(* CoDeSys 2.3 project: skv_owen1.6.pro *)
(* Title: Контроль и управление скважинами. *)
(* Version: 1.6 *)
(* Author: Пичугин А.В. *)
(* Description: Автоматизированная система контроля и управления
водонасосной станции Печорского ЛПУ МГ *)
(* Libraries: STANDARD.LIB 4.10.05 11:14:46, IECSFC.LIB 13.4.06 15:51:28, SYSLIBTIME.LIB 20.2.06 13:31:16, SysLibMem.lib 20.2.06 13:31:12, SysLibCom.lib 20.2.06 13:31:08, SYSTASKINFO.LIB 20.2.06 13:31:38, ANALYZATION.LIB 5.10.99 09:05:06, SYSLIBCALLBACK.LIB 20.2.06 13:31:08, Util.lib 18.5.10 15:14:28 *)

(* PLC configuration (modules and I/O channels)
Discrete input 8 bit [ID100] node 0, in %IB0 out %QB0 {Filtrationtime = 10; Filtrationtime = 10; Filtrationtime = 10; Filtrationtime = 10; Filtrationtime = 10; Filtrationtime = 10; Filtrationtime = 10; Filtrationtime = 10; Visibility = Yes; PinCount = 8; WatchDogPeriod = 1000; PollPeriod = 1}
  AT %IB0.0 [ByteInput] 8 discrete inputs
Discrete output - relay [ID102] node 1, in %IB1 out %QB1 {PinCount = 1; SafeValueBool = FALSE; Visibility = Yes}
  Pump4_block AT %QX1.0 [BitOutput] Блокировка насоса 4 (relay)
Discrete output - relay [ID102] node 2, in %IB2 out %QB2 {PinCount = 1; SafeValueBool = FALSE; Visibility = Yes}
  Pump5_block AT %QX2.0 [BitOutput] Блокировка насоса 5 (relay)
Discrete output - relay [ID102] node 3, in %IB3 out %QB3 {PinCount = 1; SafeValueBool = FALSE; Visibility = No}
  AT %QX3.0 [BitOutput] relay
Discrete output - relay [ID102] node 4, in %IB4 out %QB4 {PinCount = 1; SafeValueBool = FALSE; Visibility = No}
  AT %QX4.0 [BitOutput] relay
Discrete output - relay [ID102] node 5, in %IB5 out %QB5 {PinCount = 1; SafeValueBool = FALSE; Visibility = No}
  AT %QX5.0 [BitOutput] relay
Discrete output - relay [ID102] node 6, in %IB6 out %QB6 {PinCount = 1; SafeValueBool = FALSE; Visibility = No}
  AT %QX6.0 [BitOutput] relay
Special output [ID104] node 7, in %IB7 out %QB7 {Visibility = No; PinCount = 1}
  AT %QX7.0 [BitOutput] Special output
Owen (Master) [OWEN_MASTER_ID451] node 8, in %IB8 out %QB8 {Timeout = 50; Visibility = Yes}
  LError AT %QW8.0 [WordOutput] Last error
  AT %QW8.1 [WordOutput] Last hash
  LAddress AT %QW8.2 [WordOutput] Last address
  AT %QB8.3 [ComChannel] Start/Stop)
  RS-485-1 [COM1_USART] node 0, in %IB8.0 out %QB8.0 {CommunicationSpeed = 11520; Parity = NO PARITY CHECK; BitLength = 8 bits; StopLength = One stop bit; InterfaceType = RS485; FrameOriented = ASCII; Timeout = 0; Visibility = Yes}
Box_Temp AT %QD8.1.0 [FloatOutput] Температура внутренняя
Outbox_Temp AT %QD8.2.0 [FloatOutput] Температура наружная
Skv4_Temp AT %QD8.3.0 [FloatOutput] Температура внутренняя
Skv4_Level AT %QD8.4.0 [FloatOutput] Уровень воды
Skv5_Temp AT %QD8.5.0 [FloatOutput] Температура внутренняя
Skv5_Level AT %QD8.6.0 [FloatOutput] Уровень воды
Skv4_level_alarm AT %QD8.7.0 [FloatOutput] Блокировка насоса
Skv5_level_alarm AT %QD8.8.0 [FloatOutput] Блокировка насоса
Skv4_Counter AT %QD8.9.0.0 [DWordOutput] Текущее значение счетчика
Skv5_Counter AT %QD8.10.0.0 [DWordOutput] Текущее значение счетчика
Skv4_Rate AT %QD8.11.0.0 [DWordOutput] Текущее значение счетчика в физических величинах
Skv5_Rate AT %QD8.12.0.0 [DWordOutput] Текущее значение счетчика в физических величинах
Skv4_dec AT %QW8.13.0.0 [WordOutput] Положение десятичной точки умножителя
Skv5_dec AT %QW8.14.0.0 [WordOutput] Положение десятичной точки умножителя
Max_temp AT %ID9.0 [FloatInput] Максимальная температура
Min_temp AT %ID10.0 [FloatInput] Минимальная температура
Max_level AT %ID11.0 [FloatInput] Верхний аварийный уровень (ВАУ)
*)

(* Task configuration *)
TASK Alarm_control (PRIORITY := 1, INTERVAL := T#1000ms);
	Alarm_control();
END_TASK
TASK Alarm_rate_control (PRIORITY := 1, INTERVAL := T#20000ms);
	Alarm_rate_control();
END_TASK
TASK Main (PRIORITY := 1, INTERVAL := T#100ms);
	PLC_PRG();
END_TASK
TASK Terminal (PRIORITY := 1, INTERVAL := T#50ms);
	Terminal();
END_TASK

(* Global variable list: Global_Variables *)
VAR_GLOBAL RETAIN
	SMS_sPhone:ARRAY[0..4] OF STRING :='','','','','+79225830093';  				(*Номера телефонов*)
	SMS_bPhone_info:ARRAY[0..4] OF BOOL:=FALSE,FALSE,FALSE,FALSE,TRUE;		(*Отсылать ли на соотв. телефон информацию*)
	SMS_bPhone_alarm:ARRAY[0..4] OF BOOL:=FALSE,FALSE,FALSE,FALSE,TRUE;	(*Отсылать ли на соотв. телефон аварии*)
	bAlarm_old:ARRAY[0..15] OF BOOL;
	iTime_info:INT:=12; (*Время отправки информации*)
	sBalance:STRING(255);
	bRateControl:BOOL:=FALSE; (*будем считать расход?*)
END_VAR

(* Global variable list: Other *)
VAR_GLOBAL
	bAlarm:ARRAY[0..15] OF BOOL; (*Аварии текущие по 1 на каждую аварию.*)
	bAlarm_send:ARRAY[0..15] OF BOOL; (*Необходимость посылки сообщения об аварии по 1 на каждую аварию.*)
	Message:ARRAY[0..15] OF STRING; (*Сообщения о появлении или исчезновении аварий*)
	bRun:BOOL; (*Разрешение на запуск*)
	tRun:TON; (*таймер задержки начала работы*)
	(*Max_temp:REAL:=45; Максимальная температура в боксе*)
	(*Min_temp:REAL:=3; Минимальная температура в боксе*)
	rHist_temp:REAL:=1; (*Гистерезис температуры*)
	(*Max_level:REAL:=73; Верхний аварийный уровень (ВАУ)*)
	Min_level:REAL:=3; (*Нижний аварийный уровень (НАУ)*)
	rHist_level:REAL:=1; (*Гистерезис уровня*)

END_VAR

(* Global variable list: Text *)
VAR_GLOBAL
	a0:STRING:='ALARM!$0D$0A Skv4 Low Level$0D$0A Pump BLOCK $0D$0A';
	n0:STRING:='NORMA.$0D$0A Skv4 Normal Level$0D$0A Pump READY $0D$0A';
	a1:STRING:='ALARM!$0D$0A Skv5 Low Level$0D$0A Pump BLOCK $0D$0A';
	n1:STRING:='NORMA.$0D$0A Skv5 Normal Level$0D$0A Pump READY $0D$0A';
	a2:STRING:='ALARM!$0D$0A Skv4 High Level $0D$0A';
	n2:STRING:='NORMA.$0D$0A Skv4 Normal Level $0D$0A';
	a3:STRING:='ALARM!$0D$0A Skv5 High Level $0D$0A';
	n3:STRING:='NORMA.$0D$0A Skv5 Normal Level $0D$0A';
	a4:STRING:='ALARM!$0D$0A Skv4 No Flow $0D$0A';
	n4:STRING:='NORMA.$0D$0A Skv4 Flow On $0D$0A';
	n41:STRING:='NORMA.$0D$0A Skv4 Flow Off $0D$0A';
	a5:STRING:='ALARM!$0D$0A Skv5 No Flow $0D$0A';
	n5:STRING:='NORMA.$0D$0A Skv5 Flow On $0D$0A';
	n51:STRING:='NORMA.$0D$0A Skv5 Flow Off $0D$0A';
	a6:STRING:='ALARM!$0D$0A Skv4 Low Temperature $0D$0A';
	n6:STRING:='NORMA.$0D$0A Skv4 Normal Temperature $0D$0A';
	a7:STRING:='ALARM!$0D$0A Skv5 Low Temperature $0D$0A';
	n7:STRING:='NORMA.$0D$0A Skv5 Normal Temperature $0D$0A';
	a8:STRING:='ALARM!$0D$0A Box Low Temperature $0D$0A';
	n8:STRING:='NORMA.$0D$0A Box Normal Temperature $0D$0A';
	a9:STRING:='ALARM!$0D$0A Skv4 High Temperature $0D$0A';
	n9:STRING:='NORMA.$0D$0A Skv4 Normal Temperature $0D$0A';
	a10:STRING:='ALARM!$0D$0A Skv5 High Temperature $0D$0A';
	n10:STRING:='NORMA.$0D$0A Skv5 Normal Temperature $0D$0A';
	a11:STRING:='ALARM!$0D$0A Box High Temperature $0D$0A';
	n11:STRING:='NORMA.$0D$0A Box Normal Temperature $0D$0A';
	a12:STRING:='ALARM!$0D$0A Skv4 No Link $0D$0A';
	n12:STRING:='NORMA.$0D$0A Skv4 Link on $0D$0A';
	a13:STRING:='ALARM!$0D$0A Skv5 No Link $0D$0A';
	n13:STRING:='NORMA.$0D$0A Skv5 Link on $0D$0A';
	a14:STRING:='ALARM!$0D$0A Box No Link $0D$0A';
	n14:STRING:='NORMA.$0D$0A Box Link on $0D$0A';
	a15:STRING:='ALARM!$0D$0A Box No Power $0D$0A';
	n15:STRING:='NORMA.$0D$0A Box Power on $0D$0A';
END_VAR

(* POU Alarm_control, ST *)
PROGRAM Alarm_control
VAR
(*Обработка гвоздей, грызунов, монтажников, и солнечного затмения*)
	er_72: Get_Modules_Errors; (*адрес 9, ТРМ202 в боксе*)
	er_88: Get_Modules_Errors; (*адрес 11, ТРМ202 скважина 4*)
	er_104: Get_Modules_Errors; (*адрес 13, СИ30 скважина 4*)
	er_112: Get_Modules_Errors; (*адрес 14, ТРМ202 скважина 5*)
	er_128: Get_Modules_Errors; (*адрес 16, СИ30 скважина 5*)
(*Каждому модулю даем свою ошибку*)
	mod_72:BOOL:=0; (* 1 - если ошибка связи, 0 - нет *)
	mod_88:BOOL:=0;  (* 1 - если ошибка связи, 0 - нет *)
	mod_104:BOOL:=0;  (* 1 - если ошибка связи, 0 - нет *)
	mod_112:BOOL:=0;  (* 1 - если ошибка связи, 0 - нет *)
	mod_128:BOOL:=0;  (* 1 - если ошибка связи, 0 - нет *)
	hist_tempb_min:HIST;
	hist_tempb_max:HIST;
	hist_temp4_min:HIST;
	hist_temp4_max:HIST;
	hist_temp5_min:HIST;
	hist_temp5_max:HIST;
	hist_level4:HIST;
	hist_level5:HIST;
	tempb_max: BOOL;
	tempb_min: BOOL;
	temp4_max: BOOL;
	temp5_max: BOOL;
	temp5_min: BOOL;
	temp4_min: BOOL;
	level5: BOOL;
	level4: BOOL;
END_VAR
IF NOT bRun THEN
	RETURN;
END_IF

IF NOT mod_88 THEN (*если нет ошибки связи  с ТРМ202 скважина 4*)
	IF Skv4_level_alarm>0 THEN (*Проверка аварии Скв4 НАУ *)
		bAlarm[0] := TRUE;
		Message[0]:=a0;
	ELSE
		bAlarm[0] := FALSE;
		Message[0]:=n0;
	END_IF
(*-----------------------------------------------------------------------------------------------------------*)
	hist_level4(LOW:=REAL_TO_INT(Max_level-rHist_level), HIGH:=REAL_TO_INT(Max_level+rHist_level), IN:=REAL_TO_INT(Skv4_Level), OUT=>level4);
	IF  level4 THEN (*Проверка аварии Скв4 ВАУ *)
		bAlarm[2] := TRUE;
		Message[2]:=a2;
	ELSE
		bAlarm[2] := FALSE;
		Message[2]:=n2;
	END_IF
(*-----------------------------------------------------------------------------------------------------------*)
	hist_temp4_min(LOW:=REAL_TO_INT(Min_temp-rHist_temp), HIGH:=REAL_TO_INT(Min_temp+rHist_temp), IN:=REAL_TO_INT(Skv4_Temp), OUT=>temp4_min);
	IF  NOT temp4_min THEN (*Проверка аварии Скв4 темп. ниже нормы *)
		bAlarm[6] := TRUE;
		Message[6]:=a6;
	ELSE
		bAlarm[6] := FALSE;
		Message[6]:=n6;
	END_IF
(*-----------------------------------------------------------------------------------------------------------*)
	hist_temp4_max(LOW:=REAL_TO_INT(Max_temp-rHist_temp), HIGH:=REAL_TO_INT(Max_temp+rHist_temp), IN:=REAL_TO_INT(Skv4_Temp), OUT=>temp4_max);
	IF  temp4_max THEN (*Проверка аварии Скв4 темп. выше нормы *)
		bAlarm[9] := TRUE;
		Message[9]:=a9;
	ELSE
		bAlarm[9] := FALSE;
		Message[9]:=n9;
	END_IF
END_IF
(*-----------------------------------------------------------------------------------------------------------*)
(*-----------------------------------------------------------------------------------------------------------*)
IF NOT mod_112 THEN (*если нет ошибки связи  с ТРМ202 скважина 5*)
	IF Skv5_level_alarm>0 THEN  (*Проверка аварии Скв5 НАУ*)
		bAlarm[1] := TRUE;
		Message[1]:=a1;
	ELSE
		bAlarm[1] := FALSE;
		Message[1]:=n1;
	END_IF
(*-----------------------------------------------------------------------------------------------------------*)
	hist_level5(LOW:=REAL_TO_INT(Max_level-rHist_level), HIGH:=REAL_TO_INT(Max_level+rHist_level), IN:=REAL_TO_INT(Skv5_Level), OUT=>level5);
	IF level5 THEN (*Проверка аварии Скв5 ВАУ *)
		bAlarm[3] := TRUE;
		Message[3]:=a3;
	ELSE
		bAlarm[3] := FALSE;
		Message[3]:=n3;
	END_IF
(*-----------------------------------------------------------------------------------------------------------*)
	hist_temp5_min(LOW:=REAL_TO_INT(Min_temp-rHist_temp), HIGH:=REAL_TO_INT(Min_temp+rHist_temp), IN:=REAL_TO_INT(Skv5_Temp), OUT=>temp5_min);
	IF  NOT temp5_min THEN (*Проверка аварии Скв5 темп. ниже нормы *)
		bAlarm[7] := TRUE;
		Message[7]:=a7;
	ELSE
		bAlarm[7] := FALSE;
		Message[7]:=n7;
	END_IF
(*-----------------------------------------------------------------------------------------------------------*)
	hist_temp5_max(LOW:=REAL_TO_INT(Max_temp-rHist_temp), HIGH:=REAL_TO_INT(Max_temp+rHist_temp), IN:=REAL_TO_INT(Skv5_Temp), OUT=>temp5_max);
	IF   temp5_max THEN (*Проверка аварии Скв5 темп. выше нормы *)
		Message[10]:=a10;
		bAlarm[10] := TRUE;
	ELSE
		bAlarm[10] := FALSE;
		Message[10]:=n10;
	END_IF
END_IF
(*-----------------------------------------------------------------------------------------------------------*)
(*Аварии Нет протока определяются отдельно в программе Alarm_rate_control *)
(*-----------------------------------------------------------------------------------------------------------*)

IF NOT mod_72 THEN (*если нет ошибки связи  с ТРМ202 щитовая*)
	hist_tempb_min(LOW:=REAL_TO_INT(Min_temp-rHist_temp), HIGH:=REAL_TO_INT(Min_temp+rHist_temp), IN:=REAL_TO_INT(Box_Temp), OUT=>tempb_min);
	IF  NOT tempb_min THEN (*Проверка аварии Щит.  темп. ниже нормы *)
		bAlarm[8] := TRUE;
		Message[8]:=a8;
	ELSE
		bAlarm[8] := FALSE;
		Message[8]:=n8;
	END_IF
(*-----------------------------------------------------------------------------------------------------------*)
	hist_tempb_max(LOW:=REAL_TO_INT(Max_temp-rHist_temp), HIGH:=REAL_TO_INT(Max_temp+rHist_temp), IN:=REAL_TO_INT(Box_Temp), OUT=>tempb_max);
	IF  tempb_max THEN (*Проверка аварии Щит. темп. выше нормы *)
		bAlarm[11] := TRUE;
		Message[11]:=a11;
	ELSE
		bAlarm[11] := FALSE;
		Message[11]:=n11;
	END_IF
END_IF
(*-----------------------------------------------------------------------------------------------------------*)
(*-----------------------------------------------------------------------------------------------------------*)
(*Аварии Нет связи определяются  в программе Get_Modules_Errors *)
CASE LAddress OF
	72:
		er_72(err:=LError , stat=> mod_72);
	88:
		er_88(err:=LError , stat=> mod_88);
	104:
		er_104(err:=LError , stat=> mod_104);
	112:
		er_112(err:=LError , stat=> mod_112);
	128:
		er_128(err:=LError , stat=> mod_128);
END_CASE;

IF  mod_88 OR mod_104 THEN (*Проверка аварии Нет связи с скв. 4 *)
	bAlarm[12] := TRUE;
	Message[12]:=a12;
ELSE
	bAlarm[12] := FALSE;
	Message[12]:=n12;
END_IF

IF  mod_112 OR mod_128 THEN (*Проверка аварии Нет связи с скв. 5 *)
	bAlarm[13] := TRUE;
	Message[13]:=a13;
ELSE
	bAlarm[13] := FALSE;
	Message[13]:=n13;
END_IF

IF  mod_72 THEN (*Проверка аварии Нет связи с щит. *)
	bAlarm[14] := TRUE;
	Message[14]:=a14;
ELSE
	bAlarm[14] := FALSE;
	Message[14]:=n14;
END_IF

(*-----------------------------------------------------------------------------------------------------------*)
IF V220_enable=FALSE THEN  (*Проверка аварии нет питания *)
	bAlarm[15] := TRUE;
	Message[15]:=a15;
ELSE
	bAlarm[15] := FALSE;
	Message[15]:=n15;
END_IF;

(*-------------------------А теперь управляем!-------------------------------------------------*)
IF bAlarm[0] OR bAlarm[4] THEN
	Pump4_block := TRUE;
ELSE
	Pump4_block := FALSE;
END_IF
IF bAlarm[1] OR bAlarm[5] THEN
	Pump5_block := TRUE;
ELSE
	Pump5_block := FALSE;
END_IF
END_PROGRAM

(* POU Get_Modules_Errors, ST *)
FUNCTION_BLOCK Get_Modules_Errors
VAR_INPUT
	err:WORD;
END_VAR
VAR_OUTPUT
	stat:BOOL:=0;
END_VAR
VAR
	bErr:BOOL;
	rt: R_TRIG;
	tim_err: TIME := T#5s;
	t: TON;
END_VAR
IF err=81 THEN
	bErr:=TRUE;
ELSE
	bErr:=FALSE;
END_IF
(*Тригер прихода ошибки*)
rt(CLK:=bErr);
(*Если пришла ошибка, запускаем таймер*)
IF rt.Q THEN
	t(IN:=TRUE , PT:=tim_err);
END_IF
(*Вызываем таймер*)
t;
(*Если таймер не запущен и ошибки нет, то аварии нет*)
IF t.IN=FALSE AND NOT bErr THEN
	stat:=FALSE;
END_IF
(*Если таймер запущен, а ошибка ушла, то была помеха, отключаем аварию и таймер*)
IF t.IN AND err=0 THEN
	t(IN:=FALSE , PT:=tim_err);
	stat:=FALSE;
END_IF
(*Если таймер отработал, а ошибка не ушла - беда, ищем ваши гвозди ))) *)
IF t.Q THEN
	stat:=TRUE;
	t(IN:=FALSE , PT:=tim_err);
END_IF

RETURN;
END_FUNCTION_BLOCK

(* POU HIST, ST *)
FUNCTION_BLOCK HIST
VAR_INPUT
	IN:REAL;
	HIGH:REAL;
	LOW:REAL;
END_VAR
VAR_OUTPUT
	OUT:BOOL;
END_VAR
VAR
END_VAR
IF IN>HIGH THEN
	OUT:=TRUE;
END_IF
IF IN<LOW THEN
	OUT:=FALSE;
END_IF
END_FUNCTION_BLOCK

(* POU Alarm_rate_control, ST *)
PROGRAM Alarm_rate_control
VAR
	Skv4_tmp:DWORD;
	Skv5_tmp:DWORD;
END_VAR
IF NOT bRun THEN
	RETURN;
END_IF

IF bRateControl THEN
	IF Pump4_on THEN
		IF Skv4_Counter <> Skv4_tmp THEN
			bAlarm[4]:=FALSE;
			Message[4]:=n4;
			Skv4_tmp :=Skv4_Counter;
		ELSE
			bAlarm[4] := TRUE;
			Message[4]:=a4;
		END_IF;
	ELSE
		bAlarm[4] := FALSE;
		Message[4]:=n41;
		Skv4_tmp:=0;
	END_IF


	IF Pump5_on THEN
		IF Skv5_Counter <> Skv5_tmp THEN
			bAlarm[5] := FALSE;
			Message[5]:=a5;
			Skv5_tmp :=Skv5_Counter;
		ELSE
			bAlarm[5] := TRUE;
			Message[4]:=n5;
		END_IF
	ELSE
		bAlarm[5] := FALSE;
		Message[5]:=n51;
		Skv5_tmp:=0;
	END_IF
ELSE
	bAlarm[4]:= FALSE;
	bAlarm[5]:= FALSE;
END_IF
END_PROGRAM

(* POU PLC_PRG, ST *)
PROGRAM PLC_PRG
VAR
	SMS_txt: STRING(255) := '';					(*Сформированый текст СМС*)
	SMS_txt_tip:INT:=1;						(*Тип СМС. 1-аварии, 2-информация, 3-разное*)
	must_send_sms:BOOL:=FALSE;		(*Признак необходимости отправить СМС*)
	bPhone_send:ARRAY[0..4] OF BOOL:=FALSE,FALSE,FALSE,FALSE,FALSE;
	FB_SMS:GSM_Modem_SMS;
	i:INT:=0;										(*для счетчиков*)
	j:INT:=0;										(*для счетчиков*)
	jj:INT:=0;										(*для счетчиков*)
	tmp_num:STRING;
	tmp_ind:INT;
	sBalanceNum:STRING:='111';
	sBalanceText:STRING:='11';
	sBalanceCom:STRING:='AT+CUSD=1,"#100#"$0D$0A';
	com_num:PORTS:=COM1;
	sInput_command1:STRING:='Replace phone'; (*Команда смены номера телефона*)
	sInput_command2:STRING:='Alarm on'; (*Команда включения посылки аварий на телефон*)
	sInput_command3:STRING:='Alarm off'; (*Команда отключения посылки аварий на телефон*)
	sInput_command4:STRING:='Info on'; (*Команда включения посылки информации на телефон*)
	sInput_command5:STRING:='Info off'; (*Команда отключения посылки информации на телефон*)
	sInput_command6:STRING:='Get info'; (*Команда получения информации на телефон*)
	sInput_command7:STRING:='Get alarm'; (*Команда получения аварий на телефон*)
	sInput_command8:STRING:='Set time'; (*Команда установки времени отправки информации на телефоны*)
	sInput_command9:STRING:='Rate on'; (*Команда включения проверки аварии нет протока*)
	sInput_command10:STRING:='Rate off'; (*Команда выключения проверки аварии нет протока*)
	rSkv4_Rate_dec: REAL;
	rSkv5_Rate_dec: REAL;
	bInfoSended: BOOL:=FALSE; (*признак того, что информация уже отослана*)
	bBalanseQ: BOOL; (*признак запроса баланса*)
END_VAR
IF NOT bRun THEN
tRun(IN := TRUE , PT:= T#3s);
END_IF
tRun;
IF  tRun.Q THEN
	tRun(IN := FALSE, PT:= T#3s);
	SysMemSet (ADR(bAlarm_old),16#00,SIZEOF(bAlarm_old)); (*Заполняем массив отправленых аварий 0-ми, теперь все аварии станут новыми*)
	bRun:=TRUE;
END_IF
IF NOT bRun THEN
	RETURN;
END_IF


 IF must_send_sms THEN (*Если необходимо послать СМС вызываем ФБ в цикле непрерывно пока не будет выставлен выход ФБ GSM_Modem_SMS sended_OK*)
 (*********************отправляем СМС всем из списка, с учетом фильтра bPhone_send*****************************)

	CASE i OF (*перебираем телефоны*)
	0..4:	IF bPhone_send[i] AND LEN(SMS_sPhone[i])>0 THEN (*если телефону разрешено получать  и он не пустой*)
				fb_sms(com_num:=COM1,phone_num:=SMS_sPhone[i],send_SMS_text:=SMS_txt ,rcvSMS:=FALSE ); (*отправляем*)
					IF fb_sms.sended_OK THEN (*когда отправлено, переключаемся на следующий телефон*)
						IF bPhone_send[0]=TRUE THEN (*если была разрешена отправка на 0 телефон, то дальше перебирать не надо*)
							i:=255;
						ELSE
							i:=i+1;
						END_IF
					ELSE
						i:=i;
					END_IF
			ELSE (* если не разрешено, просто переключаемся на следующий телефон*)
				i:=i+1;
			END_IF
	ELSE   (* телефоны кончились, всё на родину*)
		i:=0;
		SMS_sPhone[0]:='';
		bPhone_send[0]:=FALSE; (*запрещаем посылку*)
		bPhone_send[1]:=FALSE;
		bPhone_send[2]:=FALSE;
		bPhone_send[3]:=FALSE;
		bPhone_send[4]:=FALSE;
		must_send_sms:=FALSE;


		IF  SMS_txt_tip=1 THEN
			bAlarm_old[jj]:=bAlarm[jj]; (*и отмечаем, что на аварию отреагировали*)
		END_IF
	END_CASE


(******************************************************************************************************)
(******************************************************************************************************)
ELSE (*Иначе - просто проверяем полученные  смс и следим за авариями *)


	fb_sms(com_num:=COM1,phone_num:='',send_SMS_text:='' ,rcvSMS:=TRUE );

(******************Проверяем команду на замену номера телефона***********************)
	IF FIND(fb_sms.rcvedSMS,sInput_command1)>0 THEN
		tmp_ind:=STRING_TO_INT(MID(fb_sms.rcvedSMS,1,15));
		tmp_num:=MID(fb_sms.rcvedSMS,12,17);
		IF tmp_ind>=1 AND tmp_ind<=4 THEN (*если индекс от 1 до 4, то выполняем*)
			SMS_txt:=sGetTime(0);
			SMS_txt:=CONCAT('Replace ',SMS_sPhone[tmp_ind]); (*готовим подтверждающую СМС*)
			SMS_txt:=CONCAT(SMS_txt,' on '); (*готовим*)
			SMS_txt:=CONCAT(SMS_txt,tmp_num); (*готовим*)
			SMS_txt:=CONCAT(SMS_txt,' OK '); (*готово*)
			SMS_sPhone[tmp_ind]:=tmp_num; (*меняем номер*)
		ELSE
			SMS_txt:='Error! Index mast be from 1 to 4'; (*если индекс не верен, то СМС с ошибкой*)
		END_IF
		SMS_txt_tip:=3; (*тип СМС - разное*)
		SMS_sPhone[0]:=fb_sms.rcvedPhonNum; (*номер для ответа - тот с которого пришла команда*)
		bPhone_send[0]:=TRUE;
		must_send_sms:=TRUE; (*включаем отправку*)
		RETURN; (*уходим на отправку*)
	END_IF
(******************************************************************************************************)
(******************Проверяем команду на включение посылки аварий на телефон***********************)
	IF FIND(fb_sms.rcvedSMS,sInput_command2)>0 AND iIsPhone(fb_sms.rcvedPhonNum)>0THEN
		SMS_bPhone_alarm[iIsPhone(fb_sms.rcvedPhonNum)]:=TRUE;
		SMS_txt:=CONCAT(sGetTime(0),'Set alarm on OK');
		SMS_txt_tip:=3;  (*тип СМС - разное*)
		SMS_sPhone[0]:=SMS_sPhone[iIsPhone(fb_sms.rcvedPhonNum)]; (* номер для ответа - тот с которого пришла команда*)
		bPhone_send[0]:=TRUE;
		must_send_sms:=TRUE; (*включаем отправку*)
		RETURN; (*уходим на отправку*)
	END_IF
(******************Проверяем команду на выключение посылки аварий на телефон***********************)
	IF FIND(fb_sms.rcvedSMS,sInput_command3)>0 AND iIsPhone(fb_sms.rcvedPhonNum)>0THEN
		SMS_bPhone_alarm[iIsPhone(fb_sms.rcvedPhonNum)]:=FALSE;
		SMS_txt:=CONCAT(sGetTime(0),'Set alarm off OK');
		SMS_txt_tip:=3;  (*тип СМС - разное*)
		SMS_sPhone[0]:=SMS_sPhone[iIsPhone(fb_sms.rcvedPhonNum)]; (*номер для ответа - тот с которого пришла команда*)
		bPhone_send[0]:=TRUE;
		must_send_sms:=TRUE; (*включаем отправку*)
		RETURN; (*уходим на отправку*)
	END_IF
(******************Проверяем команду на включение посылки информации на телефон***********************)
	IF FIND(fb_sms.rcvedSMS,sInput_command4)>0 AND iIsPhone(fb_sms.rcvedPhonNum)>0THEN
		SMS_bPhone_info[iIsPhone(fb_sms.rcvedPhonNum)]:=TRUE;
		SMS_txt:=CONCAT(sGetTime(0),'Set info on OK');
		SMS_txt_tip:=3;  (*тип СМС - разное*)
		SMS_sPhone[0]:=SMS_sPhone[iIsPhone(fb_sms.rcvedPhonNum)]; (*номер для ответа - тот с которого пришла команда*)
		bPhone_send[0]:=TRUE;
		must_send_sms:=TRUE; (*включаем отправку*)
		RETURN; (*уходим на отправку*)
	END_IF
(******************Проверяем команду на выключение посылки информации на телефон***********************)
	IF FIND(fb_sms.rcvedSMS,sInput_command5)>0 AND iIsPhone(fb_sms.rcvedPhonNum)>0THEN
		SMS_bPhone_info[iIsPhone(fb_sms.rcvedPhonNum)]:=FALSE;
		SMS_txt:=CONCAT(sGetTime(0),'Set info off OK');
		SMS_txt_tip:=3;  (*тип СМС - разное*)
		SMS_sPhone[0]:=SMS_sPhone[iIsPhone(fb_sms.rcvedPhonNum)]; (*номер для ответа - тот с которого пришла команда*)
		bPhone_send[0]:=TRUE;
		must_send_sms:=TRUE; (*включаем отправку*)
		RETURN; (*уходим на отправку*)
	END_IF
(******************Проверяем команду  посылки информации на телефон***********************)
	IF FIND(fb_sms.rcvedSMS,sInput_command6)>0 AND iIsPhone(fb_sms.rcvedPhonNum)>0THEN

		SMS_txt:=sGetTime(0);
		SMS_txt:=CONCAT(SMS_txt,'Skv4: ');

		SMS_txt:=CONCAT(SMS_txt,REAL_TO_STRING(Round1(Skv4_Level)));
		SMS_txt:=CONCAT(SMS_txt,'m ');
		rSkv4_Rate_dec:=Skv4_Rate/EXPT(10,Skv4_dec);
		SMS_txt:=CONCAT(SMS_txt,REAL_TO_STRING(Round1(rSkv4_Rate_dec)));
		SMS_txt:=CONCAT(SMS_txt,'m3 ');
		SMS_txt:=CONCAT(SMS_txt,REAL_TO_STRING(Round1(Skv4_Temp)));
		SMS_txt:=CONCAT(SMS_txt,'C$0D$0A');

		SMS_txt:=CONCAT(SMS_txt,'Skv5: ');
		SMS_txt:=CONCAT(SMS_txt,REAL_TO_STRING(Round1(Skv5_Level)));
		SMS_txt:=CONCAT(SMS_txt,'m ');
		rSkv5_Rate_dec:=Skv5_Rate/EXPT(10,Skv5_dec);
		SMS_txt:=CONCAT(SMS_txt,REAL_TO_STRING(Round1(rSkv5_Rate_dec)));
		SMS_txt:=CONCAT(SMS_txt,'m3 ');
		SMS_txt:=CONCAT(SMS_txt,REAL_TO_STRING(Round1(Skv5_Temp)));
		SMS_txt:=CONCAT(SMS_txt,'C$0D$0A');

		SMS_txt:=CONCAT(SMS_txt,'Box In');
		SMS_txt:=CONCAT(SMS_txt,REAL_TO_STRING(Round1(Box_Temp)));
		SMS_txt:=CONCAT(SMS_txt,'C Out');
		SMS_txt:=CONCAT(SMS_txt,REAL_TO_STRING(Round1(Outbox_Temp)));
		SMS_txt:=CONCAT(SMS_txt,'C$0D$0A');
		SMS_txt:=CONCAT(SMS_txt,'Alarms ');
		SMS_txt:=CONCAT(SMS_txt,INT_TO_STRING(iIsAlarm()));
		SMS_txt:=CONCAT(SMS_txt,'$0D$0A');
		SMS_txt:=CONCAT(SMS_txt,sBalance);
		SMS_txt_tip:=3;  (*тип СМС - разное*)
		SMS_sPhone[0]:=SMS_sPhone[iIsPhone(fb_sms.rcvedPhonNum)]; (*номер для ответа - тот с которого пришла команда*)
		bPhone_send[0]:=TRUE;
		must_send_sms:=TRUE; (*включаем отправку*)
		RETURN; (*уходим на отправку*)
	END_IF
(******************Проверяем время  посылки информации на телефон***********************)
	IF STRING_TO_INT(sGetTime(1))=iTime_info  THEN
		IF  NOT bInfoSended THEN
			SMS_txt:=sGetTime(0);
			SMS_txt:=CONCAT(SMS_txt,'Skv4: ');
			SMS_txt:=CONCAT(SMS_txt,REAL_TO_STRING(Round1(Skv4_Level)));
			SMS_txt:=CONCAT(SMS_txt,'m ');
			rSkv4_Rate_dec:=Skv4_Rate/EXPT(10,Skv4_dec);
			SMS_txt:=CONCAT(SMS_txt,REAL_TO_STRING(Round1(rSkv4_Rate_dec)));
			SMS_txt:=CONCAT(SMS_txt,'m3 ');
			SMS_txt:=CONCAT(SMS_txt,REAL_TO_STRING(Round1(Skv4_Temp)));
			SMS_txt:=CONCAT(SMS_txt,'C$0D$0A');

			SMS_txt:=CONCAT(SMS_txt,'Skv5: ');
			SMS_txt:=CONCAT(SMS_txt,REAL_TO_STRING(Round1(Skv5_Level)));
			SMS_txt:=CONCAT(SMS_txt,'m ');
			rSkv5_Rate_dec:=Skv5_Rate/EXPT(10,Skv5_dec);
			SMS_txt:=CONCAT(SMS_txt,REAL_TO_STRING(Round1(rSkv5_Rate_dec)));
			SMS_txt:=CONCAT(SMS_txt,'m3 ');
			SMS_txt:=CONCAT(SMS_txt,REAL_TO_STRING(Round1(Skv5_Temp)));
			SMS_txt:=CONCAT(SMS_txt,'C$0D$0A');

			SMS_txt:=CONCAT(SMS_txt,'Box In');
			SMS_txt:=CONCAT(SMS_txt,REAL_TO_STRING(Round1(Box_Temp)));
			SMS_txt:=CONCAT(SMS_txt,'C Out');
			SMS_txt:=CONCAT(SMS_txt,REAL_TO_STRING(Round1(Outbox_Temp)));
			SMS_txt:=CONCAT(SMS_txt,'C$0D$0A');
			SMS_txt:=CONCAT(SMS_txt,'Alarms ');
			SMS_txt:=CONCAT(SMS_txt,INT_TO_STRING(iIsAlarm()));
			SMS_txt:=CONCAT(SMS_txt,'$0D$0A');
			SMS_txt:=CONCAT(SMS_txt,sBalance);
			SMS_txt_tip:=2;  (*тип СМС - информация*)
			SMS_sPhone[0]:='';
			bPhone_send[0]:=FALSE;
			bPhone_send[1]:=SMS_bPhone_info[1];
			bPhone_send[2]:=SMS_bPhone_info[2];
			bPhone_send[3]:=SMS_bPhone_info[3];
			bPhone_send[4]:=SMS_bPhone_info[4];
			bInfoSended:=TRUE;
			must_send_sms:=TRUE; (*включаем отправку*)
		END_IF
		RETURN; (*уходим на отправку*)
	ELSE
		bInfoSended:=FALSE;
	END_IF
(******************Проверяем баланс по времени (информация-1час)***********************)
	IF STRING_TO_INT(sGetTime(1))=iTime_info-1 THEN
		IF NOT bBalanseQ THEN
			SysComWrite(com_num,ADR(sBalanceCom),LEN(sBalanceCom),0);
			bBalanseQ:=TRUE;
		END_IF
		RETURN; (*уходим на отправку*)
	ELSE
		bBalanseQ:=FALSE;
	END_IF

(******************Проверяем команду на посылку аварий на телефон***********************)
	IF FIND(fb_sms.rcvedSMS,sInput_command7)>0 AND iIsPhone(fb_sms.rcvedPhonNum)>0THEN
		SMS_sPhone[0]:=SMS_sPhone[iIsPhone(fb_sms.rcvedPhonNum)]; (*номер для ответа - тот с которого пришла команда*)
		IF iIsAlarm()=0 THEN
			SMS_txt:=CONCAT(sGetTime(0),'No Alarm');
			SMS_txt_tip:=3;  (*тип СМС - разное*)
			bPhone_send[0]:=TRUE;
			must_send_sms:=TRUE; (*включаем отправку*)
			RETURN; (*уходим на отправку*)
		ELSE
			SysMemSet (ADR(bAlarm_old),16#00,SIZEOF(bAlarm_old)); (*Заполняем массив отправленых аварий 0-ми, теперь все аварии станут новыми*)
		END_IF
	END_IF
(******************Проверяем команду на установку времени рассылки информации***********************)
	IF FIND(fb_sms.rcvedSMS,sInput_command8)>0 AND iIsPhone(fb_sms.rcvedPhonNum)>0THEN
		iTime_info:=STRING_TO_INT(MID(fb_sms.rcvedSMS,2,LEN(sInput_command8)+2));
		SMS_txt:=CONCAT(sGetTime(0),'Set time of info ');
		SMS_txt:=CONCAT(SMS_txt,INT_TO_STRING(iTime_info));
		SMS_txt:=CONCAT(SMS_txt,':00 OK');
		SMS_txt_tip:=3;  (*тип СМС - разное*)
		SMS_sPhone[0]:=SMS_sPhone[iIsPhone(fb_sms.rcvedPhonNum)]; (*номер для ответа - тот с которого пришла команда*)
		bPhone_send[0]:=TRUE;
		must_send_sms:=TRUE; (*включаем отправку*)
		RETURN; (*уходим на отправку*)
	END_IF

(******************Проверяем команду на включение проверки аварии Нет протока***********************)
	IF FIND(fb_sms.rcvedSMS,sInput_command9)>0 AND iIsPhone(fb_sms.rcvedPhonNum)>0THEN
		bRateControl:=TRUE;
		SMS_txt:=CONCAT(sGetTime(0),'Rate alarm on OK');
		SMS_txt_tip:=3;  (*тип СМС - разное*)
		SMS_sPhone[0]:=SMS_sPhone[iIsPhone(fb_sms.rcvedPhonNum)]; (*номер для ответа - тот с которого пришла команда*)
		bPhone_send[0]:=TRUE;
		must_send_sms:=TRUE; (*включаем отправку*)
		RETURN; (*уходим на отправку*)
	END_IF
(******************Проверяем команду на выключение проверки аварии Нет протока***********************)
	IF FIND(fb_sms.rcvedSMS,sInput_command10)>0 AND iIsPhone(fb_sms.rcvedPhonNum)>0THEN
		bRateControl:=FALSE;
		SMS_txt:=CONCAT(sGetTime(0),'Rate alarm off OK');
		SMS_txt_tip:=3;  (*тип СМС - разное*)
		SMS_sPhone[0]:=SMS_sPhone[iIsPhone(fb_sms.rcvedPhonNum)]; (*номер для ответа - тот с которого пришла команда*)
		bPhone_send[0]:=TRUE;
		must_send_sms:=TRUE; (*включаем отправку*)
		RETURN; (*уходим на отправку*)
	END_IF

(****************Проверяем аварии**********************************)
	CASE j OF (*перебираем аварии*)
	0..15:	bAlarm_send[j] :=bAlarm[j] XOR bAlarm_old[j];  (*Необходимо послать сообщение только об изменившихся состояниях аварий*)
			IF bAlarm_send[j] THEN
				SMS_txt:=CONCAT(sGetTime(0),Message[j]);
				bPhone_send[1]:=SMS_bPhone_alarm[1];
				bPhone_send[2]:=SMS_bPhone_alarm[2];
				bPhone_send[3]:=SMS_bPhone_alarm[3];
				bPhone_send[4]:=SMS_bPhone_alarm[4];
				SMS_txt_tip:=1;  (*тип СМС - аварии*)
				must_send_sms:=TRUE;
				jj:=j;
				j:=j+1;
			ELSE
				j:=j+1;
			END_IF
	ELSE
			j:=0;
			must_send_sms:=FALSE;
	END_CASE
(******************************************************************************************************)
END_IF
END_PROGRAM

(* POU GSM_Modem_SMS, ST *)
(*Процедура работы с GSM модемом : посылка - получение СМС*)
FUNCTION_BLOCK GSM_Modem_SMS
VAR_INPUT
	com_num:PORTS:=COM1; (*Номер порта для работы с модемом*)
	phone_num:STRING;         (*Телефонный номер для посылки смс*)
	send_SMS_text:STRING(255);           (*Строка для отправки по указанному номеру шлем если не пустая*)
	rcvSMS:BOOL;                      (*Флаг необходимости проверки SMS*)
END_VAR
VAR_OUTPUT
	rcvedSMS:STRING(255);		(*Полученное СМС*)
	rcvedPhonNum:STRING; (*Телефон с которого отправлено SMS*)
	sended_OK:BOOL;           (*Признак отправки СМС в *)
END_VAR
VAR
	port_opened: BOOL := FALSE; (*Признак открытия порта*)
	com_handle: DWORD;

(*Буферы для обмена*)
	rcvBUF: ARRAY [0..255] OF BYTE;
	rcvStr:STRING(255);
	snd_str:STRING(255);


	iter: DWORD;
	com_set: COMSETTINGS;

	sInput_command9:STRING:='Balance'; (*Признак принятого баланса*)
(*Комманда чтения СМС*)
	strGetNewSMS:STRING:='AT+CMGL="REC UNREAD"$R';
	strSetCharSet:STRING:='AT+CSCS="GSM"$R';

	strGetBalance:STRING:='AT+CUSD=1,"#100#"$R'; (*получить баланс*)
	strDelReadSMS:STRING:='AT+CMGD=1,2$R'; (*удалить все ПРОЧИТАННЫЕ и ОТПРАВЛЕННЫЕ сообщения*)
	strDelAllSMS:STRING:='AT+CMGD=1,4$R'; (*удалить все сообщения*)

	do_send_sms2: BOOL := FALSE;
	sz: DWORD := 0;
	a_char: POINTER TO STRING;
	do_rcv_sms2: BOOL := FALSE;
	port_init:BOOL:=FALSE;
	res:BOOL;

(*Таймеры ожидания для работы*)
	tmr_rcv_wait:TON;
	tmr_snd_wait:TON;
	tmr_rq_wait:TON;
END_VAR
(*Открываем порт*)
IF NOT port_opened THEN
	com_handle:=SysComOpen(com_num);
	IF com_handle<>16#FFFFFFFF THEN
		port_init:=TRUE;
	ELSE
		SysComClose(	com_num);
		com_handle:=SysComOpen(	com_num);
		port_init:=TRUE;
	END_IF

(*Настраиваем скорость*)
	com_set.Port:=com_num;
	com_set.dwBaudRate:=9600;
	com_set.byParity:=0;
	com_set.dwTimeout:=0;
	com_set.byStopBits:=0; (* *)
	com_set.dwBufferSize:=0;
	com_set.dwScan:=0;
	res:=SysComSetSettings(com_num,ADR(com_set));
(*Успешно открыли*)
	IF NOT res THEN
		port_opened:=TRUE;
		SysComWrite(com_num,ADR(strDelAllSMS),LEN(strDelAllSMS),0);
	END_IF
END_IF

(*Взводим таймер если надо*)
tmr_snd_wait(IN:=LEN(send_SMS_text)>0 AND do_send_sms2,PT:=t#5s);

(*Если таймер сработал больше не ждем ответа от модема*)
IF tmr_snd_wait.Q THEN
	do_send_sms2:=FALSE;
	tmr_snd_wait(IN:=LEN(send_SMS_text)>0 AND do_send_sms2,PT:=t#5s);
	rcvStr:='';
END_IF

(*Начинаем посылку*)
sended_OK:=FALSE;
(*Если нужно послать СМС*)
IF LEN(send_SMS_text)>0 AND NOT do_send_sms2 THEN
	snd_str:=CONCAT('AT+CMGS="',phone_num);
	snd_str:=CONCAT(snd_str,'"$R');

	SysComWrite(com_num,ADR(snd_str),LEN(snd_str),0);
	rcvStr:='';
	rcvedSMS:='';
	rcvedPhonNum:='';
(*Ждать ответа от модема*)
	do_send_sms2:=TRUE;

END_IF

(*Таймер ожидания получения*)
tmr_rcv_wait(IN:=do_rcv_sms2,PT:=t#5s);
IF tmr_rcv_wait.Q THEN
	do_rcv_sms2:=FALSE;
	tmr_rcv_wait(IN:=do_rcv_sms2,PT:=t#5s);
	rcvStr:='';
END_IF


(*Если нужно получить ответ от модема*)
IF rcvSMS AND NOT do_send_sms2 AND NOT do_rcv_sms2 THEN
	SysComWrite(com_num,ADR(strGetNewSMS),LEN(strGetNewSMS),0);
	rcvStr:='';
	do_rcv_sms2:=TRUE;
END_IF

(*Получаем данные из порта*)
sz:=SysComRead(com_num,ADR(rcvBUF),1024,0);
(*Таймер получения ответа от модема -2 секунды*)
IF LEN(rcvStr)=0 THEN
	tmr_rq_wait(IN:=FALSE,PT:=t#2s);
ELSE
	tmr_rq_wait(IN:=TRUE,PT:=t#2s);
END_IF
IF sz<>0 THEN
	(*Если данные есть то получаем строку*)
	FOR iter:=0 TO sz-1 DO
		a_char:=ADR(rcvBuf[iter]);
		rcvStr:=CONCAT(rcvStr,LEFT(a_char^,1) );
		IF LEN(rcvStr)>250 THEN
			rcvStr:=DELETE(rcvStr,1,1);
		END_IF
	END_FOR
(******************Проверяем приход баланса***********************)
	IF FIND(rcvStr,sInput_command9)<>0 THEN
		sBalance:=rcvStr; (*текст баланса*)
		sBalance:=DELETE(sBalance, FIND(rcvStr,sInput_command9)-1,1);
		sBalance:=LEFT(sBalance,LEN(sBalance)-5);
	END_IF

	IF do_send_sms2 THEN
		(*При посылке СМС ожидаем готовности модема знак >*)
		IF FIND(rcvStr,'>') <> 0 THEN
			snd_str:=send_SMS_text;
			snd_str:=CONCAT(snd_str,'$1a');
			(*Шлем SMS*)
			SysComWrite(com_num,ADR(snd_str),LEN(snd_str),0);
			do_send_sms2:=FALSE;
			(*СМС Послано*)
			sended_OK:=TRUE;
		END_IF
	END_IF
END_IF
(*Если прием СМС*)
IF do_rcv_sms2 AND tmr_rq_wait.q THEN
		(*Если ждем эхо*)
		IF FIND(rcvStr,strGetNewSMS) <> 0 THEN
			rcvStr:=DELETE(rcvStr,FIND(rcvStr,strGetNewSMS) +LEN(strGetNewSMS)+1,1);
		END_IF
		(*Начато тел. номера из россии это +7 *)
		IF FIND(rcvStr,'+7')<>0 THEN
			rcvStr:=DELETE(rcvStr,FIND(rcvStr,'+7') -1,1);
			rcvedPhonNum:=LEFT(rcvStr,FIND(rcvStr,'"')-1);
			(*СМС ограничено переводами строк*)
			rcvStr:=DELETE(rcvStr,FIND(rcvStr,'$R$N')+1,1);
			rcvedSMS:=LEFT(rcvStr,FIND(rcvStr,'$R$N')-1);
		END_IF
		rcvstr:='';
		SysComWrite(com_num,ADR(strDelReadSMS),LEN(strDelReadSMS),0);
END_IF
END_FUNCTION_BLOCK

(* POU sGetTime, ST *)
FUNCTION sGetTime : STRING
VAR_INPUT
	iTip:INT; (*Тип вывода времени. 1-часы   остальное-полностью*)
END_VAR
VAR
	GetTime: CurTimeEx;
	TimeAndDate: SystemTimeDate;
	Sys_Time: SysTime64;
	MM: UINT;
	SS: UINT;
	HH: UINT;
	D: UINT;
	M: UINT;
	Y: UINT;
END_VAR
(*********************************Текущее время**********************************)
TimeAndDate.Day :=0;
TimeAndDate.DayOfWeek :=0;
TimeAndDate.dwHighMsec :=0;
TimeAndDate.dwLowMSecs :=0;
TimeAndDate.Milliseconds :=0;
TimeAndDate.Minute :=0;
TimeAndDate.Second :=0;
TimeAndDate.Hour :=0;
TimeAndDate.Year :=0;
TimeAndDate.Month :=0;
Sys_time.ulHigh :=0;
Sys_time.ulLow :=0;
GetTime (SystemTime:=Sys_Time , TimeDate:= TimeAndDate);
CASE iTip OF
1:	sGetTime:=UINT_TO_STRING(TimeAndDate.Hour);

ELSE
sGetTime:=CONCAT(' ',UINT_TO_STRING(TimeAndDate.Day));
sGetTime:=CONCAT(sGetTime,'.');
sGetTime:=CONCAT(sGetTime,UINT_TO_STRING(TimeAndDate.Month));
sGetTime:=CONCAT(sGetTime,'.');
sGetTime:=CONCAT(sGetTime,UINT_TO_STRING(TimeAndDate.Year));
sGetTime:=CONCAT(sGetTime,'  ');
sGetTime:=CONCAT(sGetTime,UINT_TO_STRING(TimeAndDate.Hour));
sGetTime:=CONCAT(sGetTime,':');
sGetTime:=CONCAT(sGetTime,UINT_TO_STRING(TimeAndDate.Minute));
sGetTime:=CONCAT(sGetTime,':');
sGetTime:=CONCAT(sGetTime,UINT_TO_STRING(TimeAndDate.Second));
sGetTime:=CONCAT(sGetTime,' $0D$0A');
END_CASE
END_FUNCTION

(* POU iIsPhone, ST *)
FUNCTION iIsPhone : INT
VAR_INPUT
	sPhoneNum:STRING;
END_VAR
VAR
	i: INT := 1;
END_VAR
FOR i:=1 TO 4 DO
	IF sPhoneNum=SMS_sPhone[i] THEN
		iIsPhone:=i;
		RETURN;
	ELSE
		iIsPhone:=0;
	END_IF
END_FOR
END_FUNCTION

(* POU Round1, ST *)
FUNCTION Round1 : REAL
VAR_INPUT
	rNumber:REAL;
END_VAR
VAR
	rNum0:REAL;
	iNum1:INT;
	iNum2:INT;
END_VAR
rNum0:=TRUNC(rNumber*10);
iNum1:=TRUNC(rNum0*10);
iNum2:=TRUNC(rNumber*100);
IF (iNum2-iNum1)>=5 THEN
	rNum0:=rNum0+1;
ELSE
	rNum0:=rNum0;
END_IF
Round1:=rNum0/10;
END_FUNCTION

(* POU iIsAlarm, ST *)
FUNCTION iIsAlarm : INT
VAR_INPUT
END_VAR
VAR
	i:INT;
END_VAR
iIsAlarm:=0;
FOR i:=0 TO 15 DO
	IF bAlarm[i] THEN
		iIsAlarm:=iIsAlarm+1;
	END_IF
END_FOR
END_FUNCTION

(* POU Terminal, ST *)
PROGRAM Terminal
VAR
	sSend:STRING(255);
	sReciv:STRING(255);
	bSend:BOOL;
	com_num:PORTS:=COM1;
END_VAR
IF bSend THEN
sSend:=CONCAT(sSend,'$0D$0A');
SysComWrite(com_num,ADR(sSend),LEN(sSend),0);
bSend:=FALSE;
sSend:='';
END_IF
END_PROGRAM

(* Visualisation terminal
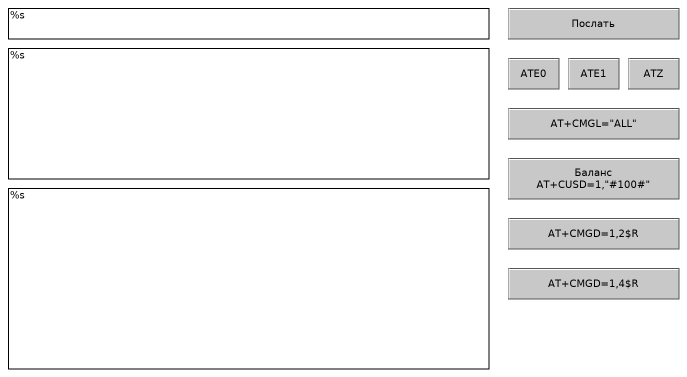
rectangle at (110,190)-(591,371): text "%s"; shows PLC_PRG.FB_SMS.rcvStr
button at (610,10)-(781,41): text "Послать"; taps Terminal.bSend
rectangle at (110,50)-(591,181): text "%s"; shows PLC_PRG.FB_SMS.snd_str
rectangle at (110,10)-(591,41): text "%s"; shows Terminal.sSend; editable
button at (610,110)-(781,141): text "AT+CMGL="ALL""; runs INTERN ASSIGN Terminal.sSend:=('AT+CMGL="ALL"')
button at (610,160)-(781,201): text "Баланс / AT+CUSD=1,"#100#""; runs INTERN ASSIGN Terminal.sSend:=('AT+CUSD=1,"#100#"')
button at (610,60)-(661,91): text "ATE0"; runs INTERN ASSIGN Terminal.sSend:=('ATE0')
button at (670,60)-(721,91): text "ATE1"; runs INTERN ASSIGN Terminal.sSend:=('ATE1')
button at (730,60)-(781,91): text "ATZ"; runs INTERN ASSIGN Terminal.sSend:=('ATZ')
button at (610,220)-(781,251): text "AT+CMGD=1,2$R"; runs INTERN ASSIGN Terminal.sSend:=('AT+CMGD=1,2$R'); tooltip удалить все ПРОЧИТАННЫЕ и ОТПРАВЛЕННЫЕ сообщения
button at (610,270)-(781,301): text "AT+CMGD=1,4$R"; runs INTERN ASSIGN Terminal.sSend:=('AT+CMGD=1,4$R'); tooltip удалить все сообщения
*)
